// TIA Portal V20 export
DATA_BLOCK "Data_State2"   // DB12
{ S7_Optimized_Access := 'FALSE' }
   VAR
      state1 : "UDT_Flowmeter_Status";
      state_2 : "UDT_Flowmeter_Stoe";
   END_VAR
BEGIN
END_DATA_BLOCK
